Fanuc KAREL source: kb00198.KL

-- PROVISIONAL review KL for V770-1; original PC SHA256 08f09a66f815ba59ff7ac126e591ad53ab9e4c90f1949e0a325bc098f75357c6
-- Incomplete behavior may be omitted. Consult companion uncertainty JSON. Do not deploy.
PROGRAM KB00198
%NOLOCKGROUP
BEGIN
  -- UNRESOLVED_PC offsets 5-14; opcodes 3F,75
  -- UNRESOLVED_PC offsets 19-26; opcodes 9D,23
  -- UNRESOLVED_PC offsets 31-38; opcodes 9D,23
  -- UNRESOLVED_PC offsets 43-79; opcodes 27,22,22,2A,22,22,22,31
  -- UNRESOLVED_PC offsets 84-88; opcodes 7F
END KB00198
